INTERFACE I_NcConveyer EXTENDS I_Conveyer

PROPERTY Axis1 : AXIS_REF
GET
END_GET
SET
END_SET
END_PROPERTY

PROPERTY Axis2 : AXIS_REF
GET
END_GET
SET
END_SET
END_PROPERTY

END_INTERFACE

(* stored: Version 1.1.0.1, ProductVersion 3.1.4024.6
   Itf I_NcConveyer: Id {117ba5e6-0593-47bb-81fe-fa0ad1622858}
   Property Axis1: Id {c71ad056-3473-4102-bd50-38f19a753c05}
   Get Get: Id {5fe67993-b685-457f-a51e-fcf9e4fa605d}
   Set Set: Id {20d840cb-3062-4686-968b-6aaf61870b25}
   Property Axis2: Id {c5b9b783-e4e1-4ff9-8f37-554ae8af245f}
   Get Get: Id {9846f172-fa37-46cf-bcf1-665672edef9c}
   Set Set: Id {d6491bc4-95f5-4c0d-b552-bbb3010796a0} *)
